FUNCTION_BLOCK OUT_TEXT (* WSTRING Output to a TextArea *)
  (* Standard: 61499-2 *)
  (* Version 0.0, 2004-06-20, Unknown, Unknown *)
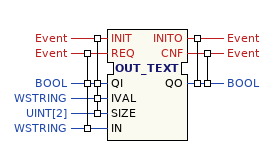
  EVENT_INPUT
    INIT WITH QI, IVAL, SIZE;
    REQ WITH QI, IN; (* Append IN to the TextArea *)
  END_EVENT
  EVENT_OUTPUT
    INITO WITH QO;
    CNF WITH QO;
  END_EVENT
  VAR_INPUT
    QI : BOOL := true;
    IVAL : WSTRING;
    SIZE : ARRAY [0..1] OF UINT := [10,20]; (* Rows,Columns *)
    IN : WSTRING;
  END_VAR
  VAR_OUTPUT
    QO : BOOL;
  END_VAR
  SERVICE OUT_TEXT/TextArea
    SEQUENCE normal_initialization
      OUT_TEXT.INIT+(IVAL) -> TextArea.initialize(IVAL) -> OUT_TEXT.INITO+(OUT);
    END_SEQUENCE
    SEQUENCE initialization_inhibited
      OUT_TEXT.INIT-() -> OUT_TEXT.INITO-();
    END_SEQUENCE
    SEQUENCE data_request
      OUT_TEXT.REQ+(IN) -> TextArea.append() -> OUT_TEXT.CNF+(OUT);
    END_SEQUENCE
    SEQUENCE not_initialized
      OUT_TEXT.REQ+() -> OUT_TEXT.CNF-();
    END_SEQUENCE
    SEQUENCE clear
      OUT_TEXT.REQ-() -> TextArea.clear() -> OUT_TEXT.CNF-();
    END_SEQUENCE
  END_SERVICE
END_FUNCTION_BLOCK
